RoboDK station: kr30 cnc 090719 6.rdk

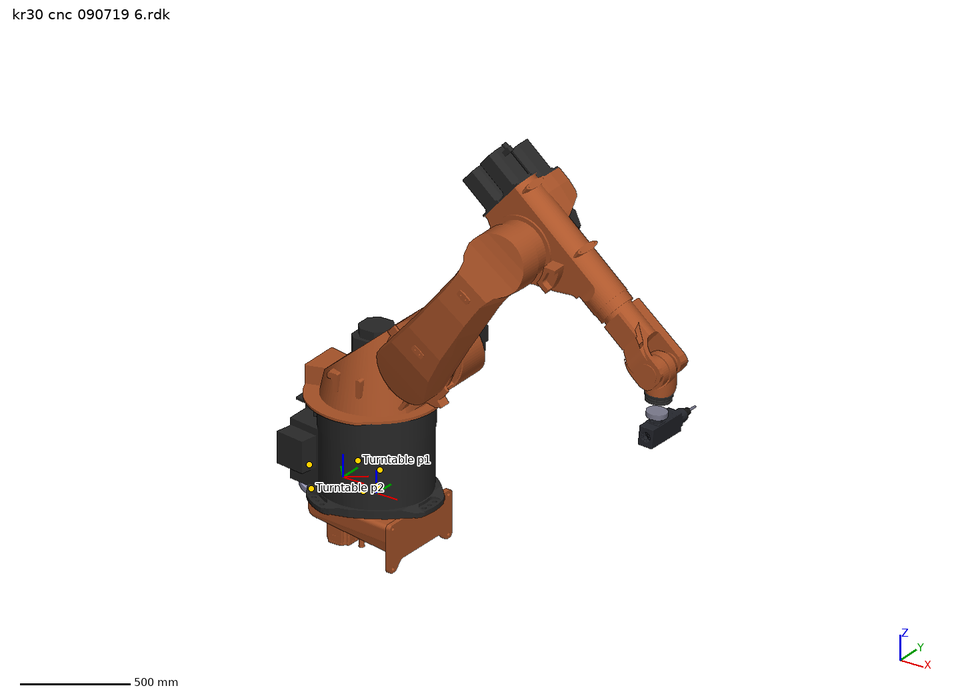
[picture v0: the station drawn from its stored meshes, robots at their saved joint values, targets as dots, program paths as lines]
Station kr30 cnc 090719 6. Poses are relative to the parent item; angles as X-Y-Z fixed-axis rotations.
  - frame GIGASHEEN 7th Axis Base at (-220, 48.2, 0) mm
    - robot KUKA KP1 MD250: 1 axes, payload 250 kg
        modified DH rows (alpha deg, a mm, theta deg, d mm): 0, 0, 0, 0
        joint limits [-3600] to [3600]; home [0]; saved at [1119.52]
      - frame Turntable Base at (0, 0, 0) mm
        - target Turntable p1 (joint target) at (82.14, 161.97, 0.25) mm, rotated rx -177.75 ry 0.19 rz 135.35 deg; joints [-0.263, -56.336, 89.398, 180.183, -62.071, -268.099] of GIGASHEEN
        - target Turntable p2 (joint target) at (-153.8, -124.05, 9.42) mm, rotated rx -178.19 ry 0.84 rz 135.28 deg; joints [-0.086, -78.923, 121.543, 181.048, -52.585, -268.908] of GIGASHEEN
        - target Turntable p3 (joint target) at (-141.11, 128.04, 4.26) mm, rotated rx -177.86 ry 2.27 rz 135.91 deg; joints [-0.629, -71.108, 99.292, 182.427, -66.433, -269.454] of GIGASHEEN
        - target Turntable p4 (joint target) at (147.86, -110.33, 4.39) mm, rotated rx -177.86 ry 2.27 rz 135.91 deg; joints [-0.623, -58.438, 110.183, 183.269, -42.9, -270.874] of GIGASHEEN
        - target Turntable p5 (joint target) at (174.66, 57.8, 0.73) mm, rotated rx -177.86 ry 2.27 rz 135.91 deg; joints [-0.699, -53.926, 95.09, 182.761, -53.469, -270.198] of GIGASHEEN
        - target Turntable p6 (joint target) at (79.99, -167.09, 6.52) mm, rotated rx -177.86 ry 2.27 rz 135.91 deg; joints [-0.573, -63.64, 117.363, 183.403, -40.923, -271] of GIGASHEEN
  - frame GIGASHEEN Base at (0, 0, 0) mm
    - robot GIGASHEEN (model KUKA KR 30 HA): 6 axes, payload 30 kg, reach 2033 mm, repeatability 0.05 mm, weight 665 kg
        modified DH rows (alpha deg, a mm, theta deg, d mm): 0, 0, 0, 815; -90, 350, 0, 0; 0, 850, -90, 0; -90, 145, 0, 820; 90, 0, 0, 0; -90, 0, 180, 170
        joint limits [-185, -135, -120, -350, -119, -350] to [185, 35, 158, 350, 119, 350]; home [0, -90, 90, 0, 0, 0]; saved at [-0.699, -53.926, 95.09, 182.761, -53.469, -270.198]
      - tool 1/2" End Mill TCP, TCP at (338.07, -0.2, 160.37) mm, rotated rx 0 ry 90 rz 0 deg, size 415.8 x 102 x 153.6 mm, geometry from GIGASHEEN
